// TIA Portal V17 program export: 1 tag tables, 1 data types, 2 data blocks, 6 code blocks (in call order from the OBs), 0 instance data blocks

VAR_GLOBAL   // PLC tag table "Default tag table"
   Start AT %M0.0 : Bool;
   Rele AT %M10.0 : Bool;
   Tag_3 AT %M0.1 : Bool;
   Stop AT %M0.2 : Bool;
   stop2 AT %M0.3 : Bool;
   tlacStartM1 AT %I0.0 : Bool;
   tlacStopM1 AT %I10.0 : Bool;
   stykM1 AT %Q0.0 : Bool;
END_VAR

TYPE "motorData"
// stored: IsFailsafeCompliant false
   STRUCT
      pocetStartu : UInt;
      otacky : Real;
      teplota : Real;
      status : Word;
   END_STRUCT;
END_TYPE

DATA_BLOCK "Global"   // DB2
{ S7_Optimized_Access := 'TRUE' }
VERSION : 0.1
// stored: AutoNumber true, DBAccessibleFromOPCUA true, DBAccessibleFromWebserver true, IsOnlyStoredInLoadMemory false, IsRetainMemResEnabled false, IsWriteProtectedInAS false, MemoryReserve 100
   VAR
      promena1 : Int;
      promena2 : DInt;
      promenou3 : DInt;
   END_VAR
BEGIN
END_DATA_BLOCK

DATA_BLOCK "Data_block_1"   // DB1
VERSION : 0.1
// stored: AutoNumber true, IsOnlyStoredInLoadMemory false, IsWriteProtectedInAS false
BEGIN
END_DATA_BLOCK

ORGANIZATION_BLOCK "Main"   // OB1, LAD, ProgramCycle
TITLE = "Main Program Sweep (Cycle)"
{ S7_Optimized_Access := 'TRUE' }
VERSION : 0.1
// stored: AutoNumber true, IsIECCheckEnabled false, SetENOAutomatically false
   VAR_INPUT
      Initial_Call : Bool;   // Initial call of this OB
      Remanence : Bool;   // =True, if remanent data are available
   END_VAR
BEGIN

REGION Network 1: ovladani M1
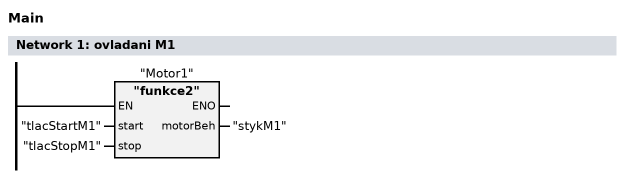
   RUNG wire#powerrail
      "Motor1"(start := "tlacStartM1", stop := "tlacStopM1", motorBeh => "stykM1")
   END_RUNG
   // the same network as SCL:
   "Motor1"(start := "tlacStartM1", stop := "tlacStopM1", motorBeh => "stykM1");   // "funkce2"
END_REGION
END_ORGANIZATION_BLOCK

FUNCTION_BLOCK "funkce2"   // FB1, LAD
{ S7_Optimized_Access := 'TRUE' }
VERSION : 0.1
// stored: AutoNumber true, IsIECCheckEnabled false, IsRetainMemResEnabled false, MemoryReserve 100, SetENOAutomatically false, UDAEnableTagReadback false
   VAR_INPUT
      start : Bool;
      stop : Bool;
   END_VAR
   VAR_OUTPUT
      motorBeh : Bool;
   END_VAR
   VAR
      statMotorBeh : Bool;
   END_VAR
   VAR_TEMP   // added for the SCL form of the ladder/FBD networks
      _w1 : Bool;
   END_VAR
BEGIN

REGION Network 1
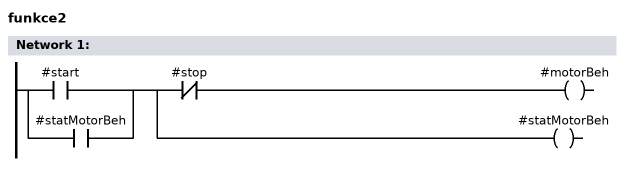
   RUNG wire#powerrail
      Contact( #start )
      wire#w1
      I_Contact( #stop )
      Coil( #motorBeh )
   END_RUNG
   RUNG wire#powerrail
      Contact( #statMotorBeh )
   END_RUNG wire#w1
   RUNG wire#w1
      Coil( #statMotorBeh )
   END_RUNG
   // the same network as SCL:
   #_w1 := #start OR #statMotorBeh;
   #motorBeh := #_w1 AND NOT #stop;
   #statMotorBeh := #_w1;
END_REGION
END_FUNCTION_BLOCK

ORGANIZATION_BLOCK "RACK_FLT"   // OB86, LAD, RackOrStationFailure
TITLE = "Loss Of Rack Fault"
VERSION : 0.1
// stored: IsIECCheckEnabled false
   VAR_TEMP
      OB86_EV_CLASS : Byte;   // 16#38/39 Event class 3
      OB86_FLT_ID : Byte;   // 16#C1/C4/C5, Fault identification code
      OB86_PRIORITY : Byte;   // Priority of OB Execution
      OB86_OB_NUMBR : Byte;   // 86 (Organization block 86, OB86)
      OB86_RESERVED_1 : Byte;   // Reserved for system
      OB86_RESERVED_2 : Byte;   // Reserved for system
      OB86_MDL_ADDR : Word;   // Base address of IM module in rack with fault
      OB86_RACKS_FLTD : Array[0..31] of Bool;   // Racks in fault
      OB86_DATE_TIME : Date_And_Time;   // Date and time OB86 started
   END_VAR
BEGIN
END_ORGANIZATION_BLOCK

ORGANIZATION_BLOCK "SYNC_1"   // OB61, LAD, SynchronousCycle
TITLE = "DP Synchronous Interrupt"
VERSION : 0.1
// stored: IsIECCheckEnabled false
   VAR_TEMP
      OB61_EV_CLASS : Byte;   // Bits 0-3 = 1 (Coming event), Bits 4-7 = 1 (Event class 1)
      OB61_STRT_INF : Byte;   // OB 61 has started
      OB61_PRIORITY : Byte;   // Priority of OB Execution
      OB61_OB_NUMBR : Byte;   // 61 (Organization block 61, OB61)
      OB61_RESERVED_1 : Byte;   // Reserved for system
      OB61_RESERVED_2 : Byte;   // Reserved for system
      OB61_GC_VIOL : Bool;   // Lost Global Control of DP system
      OB61_FIRST : Bool;   // First Execution after startup or HALT
      OB61_MISSED_EXEC : Byte;   // Count of missed executions of OB61 since it was last scheduled
      OB61_DP_ID : Byte;   // DP master system ID of the synchronous DP system
      OB61_RESERVED_3 : Byte;   // Reserved for system
      OB61_RESERVED_4 : Word;   // Reserved for system
      OB61_DATE_TIME : Date_And_Time;   // Date and time OB61 started
   END_VAR
BEGIN

REGION Network 1
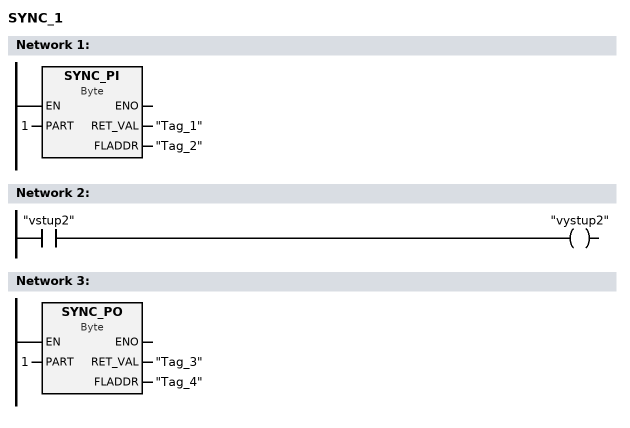
   RUNG wire#powerrail
      { S7_Templates := "value_type := Byte" } SYNC_PI(PART := 1, RET_VAL => "Tag_1", FLADDR => "Tag_2")
   END_RUNG
   // the same network as SCL:
   "Tag_1" := SYNC_PI(PART := 1, FLADDR => "Tag_2");
END_REGION

REGION Network 2
   RUNG wire#powerrail
      Contact( "vstup2" )
      Coil( "vystup2" )
   END_RUNG
   // the same network as SCL:
   "vystup2" := "vstup2";
END_REGION

REGION Network 3
   RUNG wire#powerrail
      { S7_Templates := "value_type := Byte" } SYNC_PO(PART := 1, RET_VAL => "Tag_3", FLADDR => "Tag_4")
   END_RUNG
   // the same network as SCL:
   "Tag_3" := SYNC_PO(PART := 1, FLADDR => "Tag_4");
END_REGION
END_ORGANIZATION_BLOCK

FUNCTION "funkce1" : Void   // FC1, LAD
{ S7_Optimized_Access := 'TRUE' }
AUTHOR : ziz
VERSION : 0.1
// stored: AutoNumber true, IsIECCheckEnabled false, SetENOAutomatically false, UDAEnableTagReadback false
   VAR_INPUT
      cislo1 : Int;
      cislo2 : Int;
   END_VAR
   VAR_OUTPUT
      soucet : Int;
   END_VAR
BEGIN

REGION Network 1
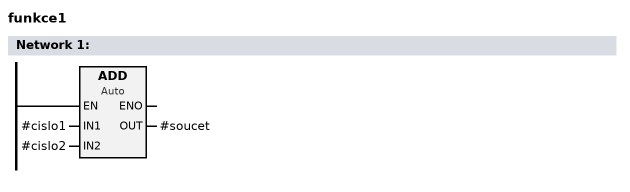
   RUNG wire#powerrail
      Add(in1 := #cislo1, in2 := #cislo2, out => #soucet)
   END_RUNG
   // the same network as SCL:
   #soucet := #cislo1 + #cislo2;
END_REGION
END_FUNCTION

FUNCTION "Block_1" : Void
{ S7_Optimized_Access := 'FALSE' }
VERSION : 0.1

BEGIN
	"xxx" := "xxx";
END_FUNCTION
